FUNCTION_BLOCK FB_ModbusSlaveRtu EXTENDS FB_UniversalModbusSlave IMPLEMENTS I_ModbusSlaveRtu
VAR
	iModbusErrorID		: MODBUS_ERRORS;// Modbus Rtu
END_VAR

bModbusError := iModbusErrorID <> MODBUSERROR_NO_ERROR;

{attribute 'monitoring' := 'variable'}
PROPERTY ModbusErrorID : MODBUS_ERRORS
GET
ModbusErrorID := iModbusErrorID;
END_GET
SET
iModbusErrorID := ModbusErrorID;
END_SET
END_PROPERTY

END_FUNCTION_BLOCK

(* stored: Version 1.1.0.1, ProductVersion 3.1.4024.12
   POU FB_ModbusSlaveRtu: Id {3c28a97a-7b9e-4799-881a-cc6e3fde9dc8}, SpecialFunc None
   Property ModbusErrorID: Id {10a0f1de-4a02-4f0a-b4da-6536bf3ef75c}
   Get Get: Id {feb78e1e-5a56-48eb-bc4b-7b331dd98e5f}
   Set Set: Id {41376bb8-baa5-43b9-b4af-8506bc2623c3} *)
